FUNCTION_BLOCK openCom (* Composite Function Block Type *)
  (* Standard: 61499-2 *)
  (* Version 0.0, 2018-03-05, 4DIAC-IDE, 4DIAC-Consortium *)
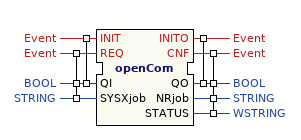
  EVENT_INPUT
    INIT WITH QI; (* Initialization Request *)
    REQ WITH QI, SYSXjob; (* Normal Execution Request *)
  END_EVENT
  EVENT_OUTPUT
    INITO WITH QO; (* Initialization Confirm *)
    CNF WITH QO, NRjob, STATUS; (* Execution Confirmation *)
  END_EVENT
  VAR_INPUT
    QI : BOOL := TRUE; (* Input event qualifier *)
    SYSXjob : STRING;
  END_VAR
  VAR_OUTPUT
    QO : BOOL; (* Output event qualifier *)
    NRjob : STRING;
    STATUS : WSTRING;
  END_VAR
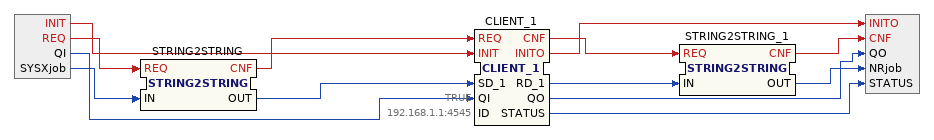
  FBS
    CLIENT_1 : CLIENT_1(QI := TRUE, ID := 192.168.1.1:4545);
    STRING2STRING : STRING2STRING;
    STRING2STRING_1 : STRING2STRING;
  END_FBS
  EVENT_CONNECTIONS
    STRING2STRING.CNF TO CLIENT_1.REQ;
    INIT TO CLIENT_1.INIT;
    REQ TO STRING2STRING.REQ;
    CLIENT_1.CNF TO STRING2STRING_1.REQ;
    STRING2STRING_1.CNF TO CNF;
    CLIENT_1.INITO TO INITO;
  END_CONNECTIONS
  DATA_CONNECTIONS
    SYSXjob TO STRING2STRING.IN;
    STRING2STRING.OUT TO CLIENT_1.SD_1;
    CLIENT_1.RD_1 TO STRING2STRING_1.IN;
    CLIENT_1.QO TO QO;
    STRING2STRING_1.OUT TO NRjob;
    CLIENT_1.STATUS TO STATUS;
    QI TO CLIENT_1.QI;
  END_CONNECTIONS
END_FUNCTION_BLOCK
